// TIA Portal project "practica3_1_3" (V14)

(* hardware
DEVICE "S71500/ET200MP station_1"  S7-1500 station
   slot 0: "Perfil soporte_0"  Rack  6ES7 590-1***0-0AA0
   slot 1: "PLC_1"  CPU 1512C-1 PN  6ES7 512-1CK00-0AB0  V2.1
      slot 3: "Display de la CPU_1"  6ES7591-1AA00-0AA0
DEVICE "PC-System_1"  SIMATIC PC station
   slot 0: "Estación PC SIMATIC"  Rail  SIMATIC PC-Station  V1.0
      slot 125: "Stationmanager"  Station_Manager  V6.0.4
   slot 1: "HMI_RT_1"  WinCC RT Advanced  6AV2 104-0xxxx-xxxx  14.0.0.0
      slot 33792: "Interfaz host"  Host interface
   slot 2: "IE general_1"  IE General  IE_CP  V8.2.0
*)

// ===== PLC "PLC_1"  CPU 1512C-1 PN =====

VAR_GLOBAL   // PLC tag table "Tabla de variables estándar"
   "Tag_1" AT %IW64 : Int;
   "Tag_2" AT %MD100 : Real;
   "PT100" AT %MD102 : Real;
   "setopoint" AT %MW56 : Int;
   "Tag_5" AT %Q4.0 : Bool;
   "Start" AT %M0.0 : Bool;
   "Stop" AT %M0.1 : Bool;
   "activarpid1" AT %M0.2 : Bool;
   "activarpid2" AT %M0.3 : Bool;
   "activarpid3" AT %M0.4 : Bool;
   "activarpid4" AT %M0.5 : Bool;
   "activacion1" AT %M0.6 : Bool;
   "activacion2" AT %M0.7 : Bool;
   "activacion3" AT %M1.0 : Bool;
   "actvacion4" AT %M1.1 : Bool;
   "temp1" AT %MD2 : DInt;
   "rangomaxT1" AT %MD6 : DInt;
   "rangominT1" AT %MD10 : DInt;
   "PT100Dint" AT %MD14 : DInt;
   "temp2" AT %MD18 : DInt;
   "rangomaxT2" AT %MD22 : DInt;
   "rangominT2" AT %MD26 : DInt;
   "temp3" AT %MD30 : DInt;
   "rangomaxT3" AT %MD34 : DInt;
   "rangominT3" AT %MD38 : DInt;
   "temp4" AT %MD42 : DInt;
   "rangomaxT4" AT %MD46 : DInt;
   "rangominT4" AT %MD50 : DInt;
   "auxsecuencia1" AT %MW54 : Int;
   "auxsecuencia2" AT %MW58 : Int;
   "Tag_3" AT %IW6 : Int;
   "Tag_4" AT %IW126 : Int;
   "Tag_6" AT %IW132 : Int;
   "Tag_7" AT %IW134 : Int;
   "Tag_8" AT %MW200 : Int;
END_VAR

DATA_BLOCK "Variables de tiempo"   // DB2
{ S7_Optimized_Access := 'TRUE' }
VERSION : 0.1
   VAR RETAIN
      TiempoP1 : DInt := 1000;
      TiempoP2 : DInt := 1000;
      TiempoP3 : DInt := 1000;
      TiempoP4 : DInt := 1000;
      Tempe_etapa1 : DInt := 20;
      Tempe_etapa2 : DInt := 20;
      Tempe_etapa3 : DInt := 20;
      Tempe_etapa4 : DInt := 20;
   END_VAR
   VAR
      Nombre : String := 'Seleccione la receta';
   END_VAR
BEGIN
END_DATA_BLOCK

DATA_BLOCK "secuencia_DB"   // DB3
{ S7_Optimized_Access := 'TRUE' }
VERSION : 0.1
// stored: InstanceOfName secuencia
"secuencia"
BEGIN
END_DATA_BLOCK

DATA_BLOCK "Reloj"   // DB4
{ S7_Optimized_Access := 'TRUE' }
VERSION : 0.1
   VAR
      Hora_actual : DTL;
   END_VAR
   VAR RETAIN
      Ajustar_hora : DTL;
   END_VAR
   VAR
      Estado_lectura : Word;
      Escribir_hora : Bool;
      Estado_escritura : Word;
   END_VAR
   VAR RETAIN
      Gain_1 : Real;
      Ti : Real;
      Td : Real;
      TdFiltRatio : Real;
      PWeighting : Real;
      DWeighting : Real;
      Cycle : Real;
   END_VAR
BEGIN
END_DATA_BLOCK

FUNCTION_BLOCK "secuencia"   // FB1, GRAPH_PLUS
{ S7_Optimized_Access := 'TRUE' }
VERSION : 0.1
   VAR_INPUT
      OFF_SQ : Bool := false;   // Desactivar cadena
      INIT_SQ : Bool := false;   // Poner cadena en estado inicial
      ACK_EF : Bool := false;   // Acusar todos los errores y fallos
      S_PREV : Bool := false;   // Mostrar la etapa anterior en el parámetro S_NO
      S_NEXT : Bool := false;   // Mostrar la etapa siguiente en el parámetro S_NO
      SW_AUTO : Bool := false;   // Modo automático
      SW_TAP : Bool := false;   // Semiautomático/continuar con transición
      SW_TOP : Bool := false;   // Semiautomático/transición ignorada
      SW_MAN : Bool := false;   // Modo manual
      S_SEL : Int := 0;   // Seleccionar la etapa que debe mostrarse en S_NO
      S_ON : Bool := false;   // Activar la etapa del parámetro S_NO
      S_OFF : Bool := false;   // Desactivar el incremento presente en el parámetro S_NO
      T_PUSH : Bool := false;   // Habilitar conmutación de transición en modo semiautomático
   END_VAR
   VAR_OUTPUT
      S_NO : Int := 0;   // Número de etapa
      S_MORE : Bool := false;   // Existen más etapas que pueden mostrarse en S_NO.
      S_ACTIVE : Bool := false;   // El incremento presente en el parámetro S_NO está activo
      ERR_FLT : Bool := false;   // Error de grupo interlock o supervisión
      AUTO_ON : Bool := false;   // Modo automático activado
      TAP_ON : Bool := false;   // Modo semiautomático/etapa con transición activada
      TOP_ON : Bool := false;   // Modo semiautomático/Ignorar transición activado
      MAN_ON : Bool := false;   // Modo manual activado
   END_VAR
   VAR
      HMI_INFO : Array[0..8] of UInt;
      IF_PAR : G7_IfParPlus_V4;
      RT_DATA : G7_RTDataPlus_V4;   // Área de datos interna
      Trans2 : G7_TransitionPlus_V4;   // Estructura de la transición
      Trans3 : G7_TransitionPlus_V4;   // Estructura de la transición
      Trans4 : G7_TransitionPlus_V4;   // Estructura de la transición
      Trans5 : G7_TransitionPlus_V4;   // Estructura de la transición
      Trans11 : G7_TransitionPlus_V4;   // Estructura de la transición
      Trans12 : G7_TransitionPlus_V4;   // Estructura de la transición
      Trans13 : G7_TransitionPlus_V4;   // Estructura de la transición
      Trans14 : G7_TransitionPlus_V4;   // Estructura de la transición
      Trans15 : G7_TransitionPlus_V4;   // Estructura de la transición
      reposo : G7_StepPlus_V4;   // Estructura de la etapa
      "Etapa 1" : G7_StepPlus_V4;   // Estructura de la etapa
      "Etapa 2" : G7_StepPlus_V4;   // Estructura de la etapa
      "Etapa 3" : G7_StepPlus_V4;   // Estructura de la etapa
      "paso 4" : G7_StepPlus_V4;   // Estructura de la etapa
      "Verificación Sp" : G7_StepPlus_V4;   // Estructura de la etapa
      Verificación_Et2 : G7_StepPlus_V4;   // Estructura de la etapa
      Verificación_Et3 : G7_StepPlus_V4;   // Estructura de la etapa
      "Verificación Et_4" : G7_StepPlus_V4;   // Estructura de la etapa
      SINI : Array[0..1] of USInt;
      LSTT : Array[0..8] of USInt;
      ATAJ : Array[0..8] of USInt;
      ATAB : Array[0..8] of USInt;
      PSTT : Array[0..8] of USInt;
      NSTT : Array[0..8] of USInt;
      ASSJ : Array[0..8] of USInt;
      ASSB : Array[0..8] of USInt;
      PTTS : Array[0..8] of USInt;
      NTTS : Array[0..8] of USInt;
      SW_SQTS : Array[0..8] of USInt;
      SWITCH : Array[0..0] of USInt;
      TVX : Array[0..1] of USInt;
      TTX : Array[0..1] of USInt;
      TSX : Array[0..1] of USInt;
      S00X : Array[0..1] of USInt;
      SOFFX : Array[0..1] of USInt;
      SONX : Array[0..1] of USInt;
      SAX : Array[0..1] of USInt;
      SERRX : Array[0..9] of USInt;
      SMX : Array[0..9] of USInt;
      S0X : Array[0..9] of USInt;
      S1X : Array[0..9] of USInt;
      IL_ALARM_INST : Diag_Alarm;
      SUP_ALARM_INST : Diag_Alarm;
      STEP_TIME_ALARM_INST : Diag_Alarm;
      IEC_TIMER_INST : IEC_TIMER;
   END_VAR
   // SINI[0] := 2;
   // LSTT[0] := 255;
   // LSTT[1] := 255;
   // LSTT[2] := 255;
   // LSTT[8] := 255;
   // ATAJ[1] := 1;
   // ATAJ[2] := 2;
   // ATAJ[3] := 3;
   // ATAJ[4] := 4;
   // ATAJ[5] := 5;
   // ATAJ[6] := 6;
   // ATAJ[7] := 7;
   // ATAJ[8] := 8;
   // ATAB[1] := 1;
   // ATAB[2] := 2;
   // ATAB[3] := 3;
   // NSTT[6] := 2;
   // ATAB[5] := 5;
   // ATAB[6] := 6;
   // ATAB[7] := 7;
   // ATAB[8] := 8;
   // PSTT[1] := 2;
   // PSTT[2] := 3;
   // PSTT[3] := 4;
   // PSTT[8] := 8;
   // PSTT[5] := 5;
   // PSTT[6] := 6;
   // PSTT[7] := 7;
   // NSTT[5] := 1;
   // NSTT[0] := 6;
   // NSTT[1] := 7;
   // NSTT[2] := 8;
   // NSTT[8] := 4;
   // ASSJ[1] := 1;
   // ASSJ[2] := 2;
   // ASSJ[3] := 3;
   // ASSJ[4] := 4;
   // ASSB[1] := 1;
   // ASSB[2] := 2;
   // ASSB[3] := 3;
   // ASSB[4] := 4;
   // PTTS[0] := 255;
   // PTTS[5] := 4;
   // PTTS[3] := 7;
   // PTTS[4] := 8;
   // NTTS[5] := 5;
   // NTTS[2] := 1;
   // NTTS[3] := 2;
   // NTTS[4] := 3;
   // TVX[0] := 16#1;
   // TTX[0] := 16#1;
   // TSX[0] := 16#1;
   // S00X[0] := 16#1;
   // SOFFX[0] := 16#1;
   // SONX[0] := 16#1;
   // SAX[0] := 16#1;
   // SERRX[0] := 16#1;
   // SMX[0] := 16#1;
   // S0X[0] := 16#1;
   // S1X[0] := 16#1;
   // LSTT[4] := 255;
   // NSTT[7] := 3;
   // ATAB[4] := 4;
   // PSTT[0] := 1;
   // NSTT[4] := 5;
   // ASSJ[5] := 5;
   // ASSB[5] := 5;
   // PTTS[1] := 5;
   // NTTS[0] := 4;
   // LSTT[5] := 255;
   // LSTT[6] := 255;
   // LSTT[7] := 255;
   // ASSJ[6] := 6;
   // ASSJ[7] := 7;
   // ASSJ[8] := 8;
   // ASSB[6] := 6;
   // ASSB[7] := 7;
   // ASSB[8] := 8;
   // PTTS[2] := 6;
   // PTTS[7] := 1;
   // PTTS[8] := 2;
   // NTTS[6] := 6;
   // NTTS[7] := 7;
   // NTTS[8] := 8;
BEGIN
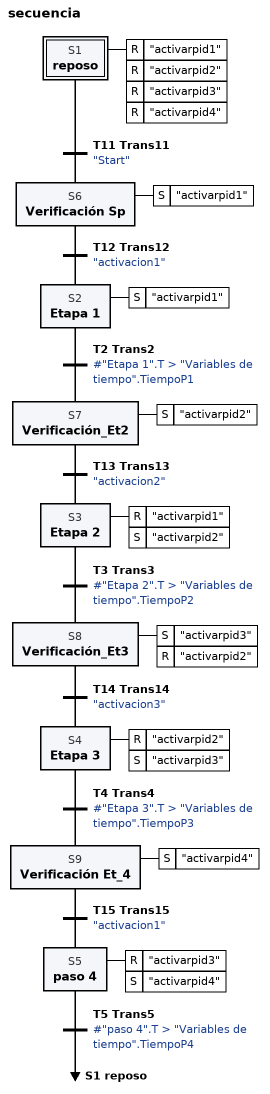
   // sequencer 1
   INITIAL_STEP reposo:   // S1, max time T#10S, warning time T#7S
              R    "activarpid1"
              R    "activarpid2"
              R    "activarpid3"
              R    "activarpid4"
   END_STEP
   TRANSITION Trans11 FROM reposo TO "Verificación Sp"   // T11
      := "Start";
   END_TRANSITION
   STEP "Etapa 1":   // S2, max time T#10S, warning time T#7S
              S    "activarpid1"
   END_STEP
   TRANSITION Trans2 FROM "Etapa 1" TO Verificación_Et2   // T2
      := #"Etapa 1".T > "Variables de tiempo".TiempoP1;
   END_TRANSITION
   STEP "Etapa 2":   // S3, max time T#10S, warning time T#7S
              R    "activarpid1"
              S    "activarpid2"
   END_STEP
   TRANSITION Trans3 FROM "Etapa 2" TO Verificación_Et3   // T3
      := #"Etapa 2".T > "Variables de tiempo".TiempoP2;
   END_TRANSITION
   STEP "Etapa 3":   // S4, max time T#10S, warning time T#7S
              R    "activarpid2"
              S    "activarpid3"
   END_STEP
   TRANSITION Trans4 FROM "Etapa 3" TO "Verificación Et_4"   // T4
      := #"Etapa 3".T > "Variables de tiempo".TiempoP3;
   END_TRANSITION
   STEP "paso 4":   // S5, max time T#10S, warning time T#7S
              R    "activarpid3"
              S    "activarpid4"
   END_STEP
   TRANSITION Trans5 FROM "paso 4" TO reposo   // T5, jump
      := #"paso 4".T > "Variables de tiempo".TiempoP4;
   END_TRANSITION
   STEP "Verificación Sp":   // S6, max time T#10S, warning time T#7S
              S    "activarpid1"
   END_STEP
   TRANSITION Trans12 FROM "Verificación Sp" TO "Etapa 1"   // T12
      := "activacion1";
   END_TRANSITION
   STEP Verificación_Et2:   // S7, max time T#10S, warning time T#7S
              S    "activarpid2"
   END_STEP
   TRANSITION Trans13 FROM Verificación_Et2 TO "Etapa 2"   // T13
      := "activacion2";
   END_TRANSITION
   STEP Verificación_Et3:   // S8, max time T#10S, warning time T#7S
              S    "activarpid3"
              R    "activarpid2"
   END_STEP
   TRANSITION Trans14 FROM Verificación_Et3 TO "Etapa 3"   // T14
      := "activacion3";
   END_TRANSITION
   STEP "Verificación Et_4":   // S9, max time T#10S, warning time T#7S
              S    "activarpid4"
   END_STEP
   TRANSITION Trans15 FROM "Verificación Et_4" TO "paso 4"   // T15
      := "activacion1";
   END_TRANSITION
END_FUNCTION_BLOCK

FUNCTION "normalizar_temp" : Void   // FC1, LAD
{ S7_Optimized_Access := 'TRUE' }
VERSION : 0.1
BEGIN

REGION Network 1: Ajuste de los datos de entrada
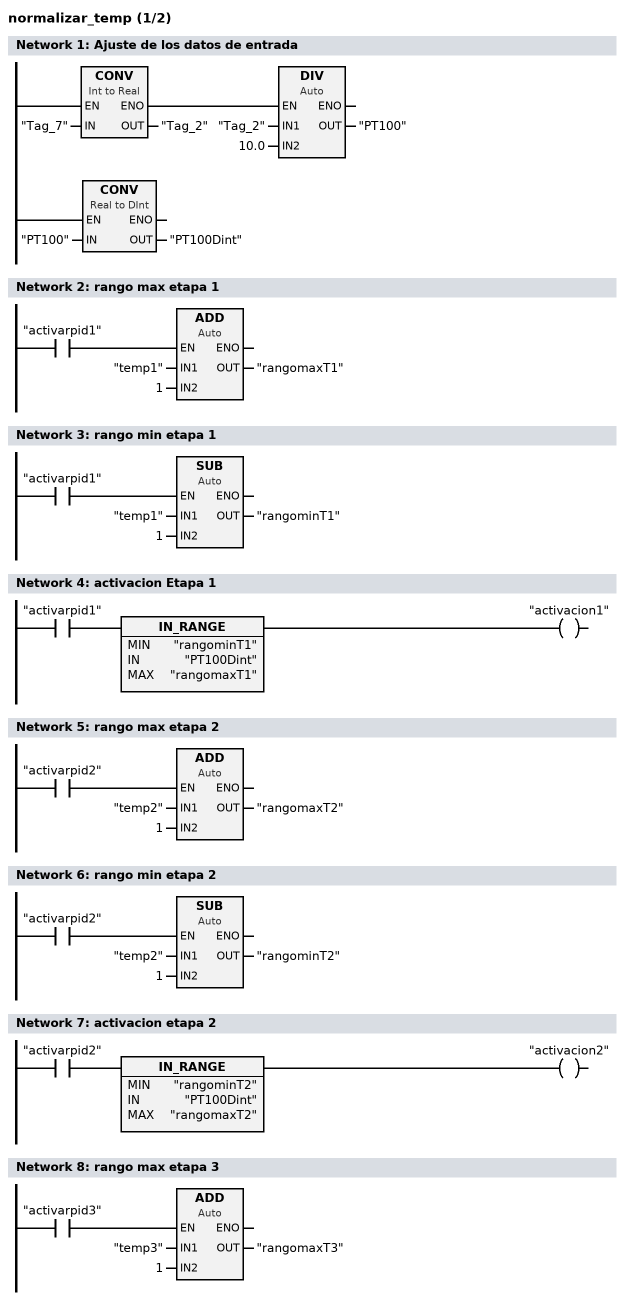
   RUNG wire#powerrail
      { S7_Templates := "[SrcType := Int, DestType := Real]" } Convert(in := "Tag_7", out => "Tag_2")
      Div(in1 := "Tag_2", in2 := 10.0, out => "PT100")
   END_RUNG
   RUNG wire#powerrail
      { S7_Templates := "[SrcType := Real, DestType := DInt]" } Convert(in := "PT100", out => "PT100Dint")
   END_RUNG
   // the same network as SCL:
   "Tag_2" := INT_TO_REAL("Tag_7");
   "PT100" := "Tag_2" / 10.0;
   "PT100Dint" := REAL_TO_DINT("PT100");
END_REGION

REGION Network 2: rango max etapa 1
   RUNG wire#powerrail
      Contact( "activarpid1" )
      Add(in1 := "temp1", in2 := 1, out => "rangomaxT1")
   END_RUNG
   // the same network as SCL:
   IF "activarpid1" THEN "rangomaxT1" := "temp1" + 1; END_IF;
END_REGION

REGION Network 3: rango min etapa 1
   RUNG wire#powerrail
      Contact( "activarpid1" )
      Sub(in1 := "temp1", in2 := 1, out => "rangominT1")
   END_RUNG
   // the same network as SCL:
   IF "activarpid1" THEN "rangominT1" := "temp1" - 1; END_IF;
END_REGION

REGION Network 4: activacion Etapa 1
   RUNG wire#powerrail
      Contact( "activarpid1" )
      { S7_Templates := "SrcType := DInt" } InRange(min := "rangominT1", in := "PT100Dint", max := "rangomaxT1")
      Coil( "activacion1" )
   END_RUNG
   // the same network as SCL:
   "activacion1" := "activarpid1" AND ("rangominT1" <= "PT100Dint") AND ("PT100Dint" <= "rangomaxT1");
END_REGION

REGION Network 5: rango max etapa 2
   RUNG wire#powerrail
      Contact( "activarpid2" )
      Add(in1 := "temp2", in2 := 1, out => "rangomaxT2")
   END_RUNG
   // the same network as SCL:
   IF "activarpid2" THEN "rangomaxT2" := "temp2" + 1; END_IF;
END_REGION

REGION Network 6: rango min etapa 2
   RUNG wire#powerrail
      Contact( "activarpid2" )
      Sub(in1 := "temp2", in2 := 1, out => "rangominT2")
   END_RUNG
   // the same network as SCL:
   IF "activarpid2" THEN "rangominT2" := "temp2" - 1; END_IF;
END_REGION

REGION Network 7: activacion etapa 2
   RUNG wire#powerrail
      Contact( "activarpid2" )
      { S7_Templates := "SrcType := DInt" } InRange(min := "rangominT2", in := "PT100Dint", max := "rangomaxT2")
      Coil( "activacion2" )
   END_RUNG
   // the same network as SCL:
   "activacion2" := "activarpid2" AND ("rangominT2" <= "PT100Dint") AND ("PT100Dint" <= "rangomaxT2");
END_REGION

REGION Network 8: rango max etapa 3
   RUNG wire#powerrail
      Contact( "activarpid3" )
      Add(in1 := "temp3", in2 := 1, out => "rangomaxT3")
   END_RUNG
   // the same network as SCL:
   IF "activarpid3" THEN "rangomaxT3" := "temp3" + 1; END_IF;
END_REGION

REGION Network 9: rango min paso 3
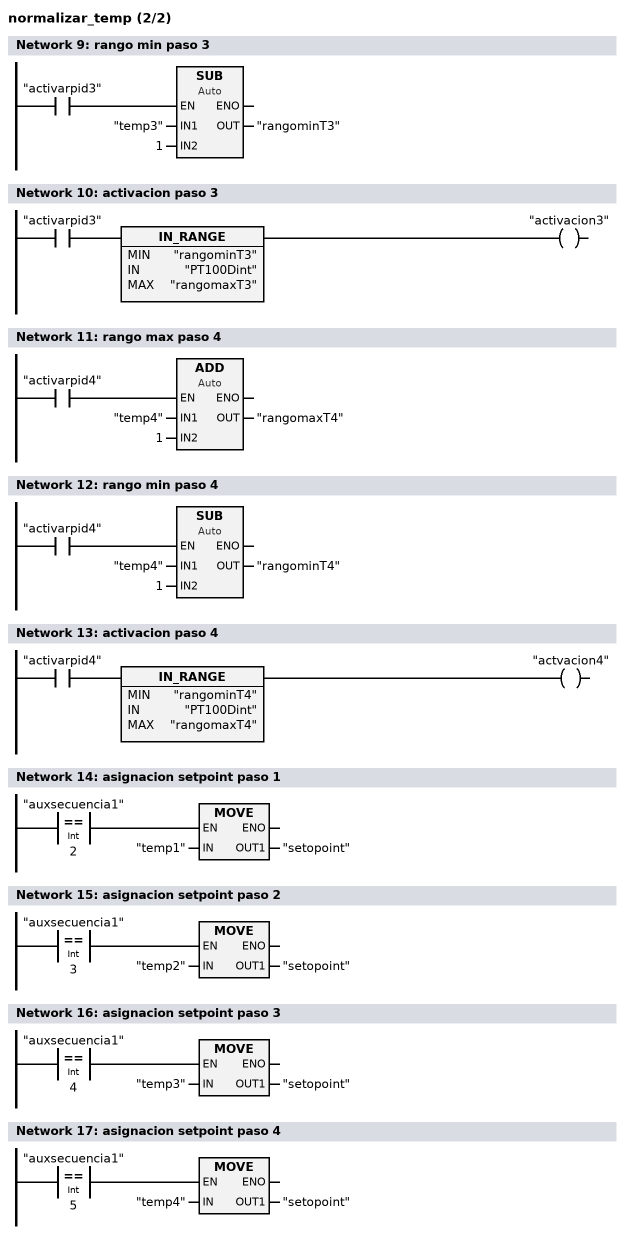
   RUNG wire#powerrail
      Contact( "activarpid3" )
      Sub(in1 := "temp3", in2 := 1, out => "rangominT3")
   END_RUNG
   // the same network as SCL:
   IF "activarpid3" THEN "rangominT3" := "temp3" - 1; END_IF;
END_REGION

REGION Network 10: activacion paso 3
   RUNG wire#powerrail
      Contact( "activarpid3" )
      { S7_Templates := "SrcType := DInt" } InRange(min := "rangominT3", in := "PT100Dint", max := "rangomaxT3")
      Coil( "activacion3" )
   END_RUNG
   // the same network as SCL:
   "activacion3" := "activarpid3" AND ("rangominT3" <= "PT100Dint") AND ("PT100Dint" <= "rangomaxT3");
END_REGION

REGION Network 11: rango max paso 4
   RUNG wire#powerrail
      Contact( "activarpid4" )
      Add(in1 := "temp4", in2 := 1, out => "rangomaxT4")
   END_RUNG
   // the same network as SCL:
   IF "activarpid4" THEN "rangomaxT4" := "temp4" + 1; END_IF;
END_REGION

REGION Network 12: rango min paso 4
   RUNG wire#powerrail
      Contact( "activarpid4" )
      Sub(in1 := "temp4", in2 := 1, out => "rangominT4")
   END_RUNG
   // the same network as SCL:
   IF "activarpid4" THEN "rangominT4" := "temp4" - 1; END_IF;
END_REGION

REGION Network 13: activacion paso 4
   RUNG wire#powerrail
      Contact( "activarpid4" )
      { S7_Templates := "SrcType := DInt" } InRange(min := "rangominT4", in := "PT100Dint", max := "rangomaxT4")
      Coil( "actvacion4" )
   END_RUNG
   // the same network as SCL:
   "actvacion4" := "activarpid4" AND ("rangominT4" <= "PT100Dint") AND ("PT100Dint" <= "rangomaxT4");
END_REGION

REGION Network 14: asignacion setpoint paso 1
   RUNG wire#powerrail
      { S7_Templates := "SrcType := Int" } EQ_Contact(in1 := "auxsecuencia1", in2 := 2)
      Move(in := "temp1", out1 => "setopoint")
   END_RUNG
   // the same network as SCL:
   IF "auxsecuencia1" = 2 THEN "setopoint" := "temp1"; END_IF;
END_REGION

REGION Network 15: asignacion setpoint paso 2
   RUNG wire#powerrail
      { S7_Templates := "SrcType := Int" } EQ_Contact(in1 := "auxsecuencia1", in2 := 3)
      Move(in := "temp2", out1 => "setopoint")
   END_RUNG
   // the same network as SCL:
   IF "auxsecuencia1" = 3 THEN "setopoint" := "temp2"; END_IF;
END_REGION

REGION Network 16: asignacion setpoint paso 3
   RUNG wire#powerrail
      { S7_Templates := "SrcType := Int" } EQ_Contact(in1 := "auxsecuencia1", in2 := 4)
      Move(in := "temp3", out1 => "setopoint")
   END_RUNG
   // the same network as SCL:
   IF "auxsecuencia1" = 4 THEN "setopoint" := "temp3"; END_IF;
END_REGION

REGION Network 17: asignacion setpoint paso 4
   RUNG wire#powerrail
      { S7_Templates := "SrcType := Int" } EQ_Contact(in1 := "auxsecuencia1", in2 := 5)
      Move(in := "temp4", out1 => "setopoint")
   END_RUNG
   // the same network as SCL:
   IF "auxsecuencia1" = 5 THEN "setopoint" := "temp4"; END_IF;
END_REGION
END_FUNCTION

FUNCTION "Lectura hora" : Void   // FC2, LAD
{ S7_Optimized_Access := 'TRUE' }
VERSION : 0.1
BEGIN

REGION Network 1: leer hora
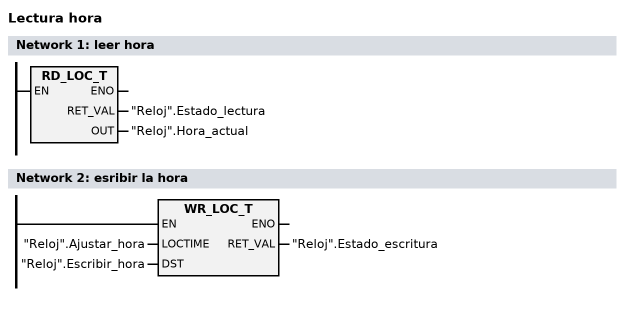
   "Reloj".Estado_lectura := RD_LOC_T(OUT => "Reloj".Hora_actual);
END_REGION

REGION Network 2: esribir la hora
   "Reloj".Estado_escritura := WR_LOC_T(LOCTIME := "Reloj".Ajustar_hora, DST := "Reloj".Escribir_hora);
END_REGION
END_FUNCTION

ORGANIZATION_BLOCK "Main"   // OB1, LAD, ProgramCycle
TITLE = "Main Program Sweep (Cycle)"
{ S7_Optimized_Access := 'TRUE' }
VERSION : 0.1
   VAR_INPUT
      Initial_Call : Bool;   // Initial call of this OB
      Remanence : Bool;   // =True, if remanent data are available
   END_VAR
BEGIN

REGION Network 1
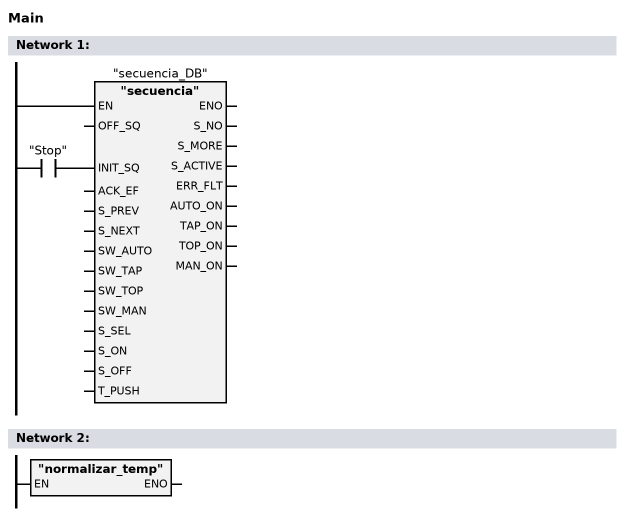
   RUNG wire#powerrail
      "secuencia_DB"(INIT_SQ := wire#w1, OFF_SQ :=, ACK_EF :=, S_PREV :=, S_NEXT :=, SW_AUTO :=, SW_TAP :=, SW_TOP :=, SW_MAN :=, S_SEL :=, S_ON :=, S_OFF :=, T_PUSH :=, S_NO =>, S_MORE =>, S_ACTIVE =>, ERR_FLT =>, AUTO_ON =>, TAP_ON =>, TOP_ON =>, MAN_ON =>)
   END_RUNG
   RUNG wire#powerrail
      Contact( "Stop" )
   END_RUNG wire#w1
   // the same network as SCL:
   "secuencia_DB"(INIT_SQ := "Stop");   // "secuencia"
END_REGION

REGION Network 2
   RUNG wire#powerrail
      "normalizar_temp"()
   END_RUNG
   // the same network as SCL:
   "normalizar_temp"();
END_REGION
END_ORGANIZATION_BLOCK

ORGANIZATION_BLOCK "Cyclic interrupt"   // OB30, LAD, CyclicInterrupt
{ S7_Optimized_Access := 'TRUE' }
VERSION : 0.1
   VAR_INPUT
      Initial_Call : Bool;   // Initial call of this OB
      Event_Count : Int;   // Events discarded
   END_VAR
BEGIN

REGION Network 1
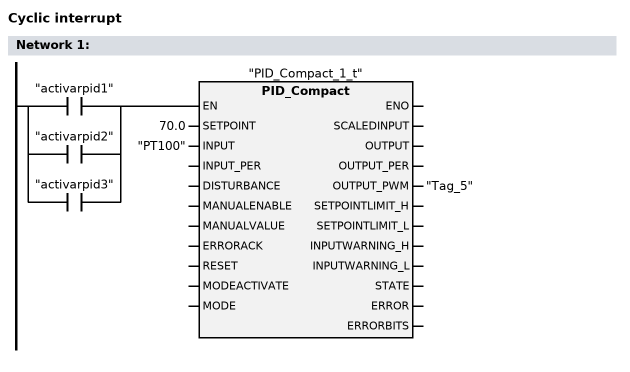
   IF "activarpid1" OR "activarpid2" OR "activarpid3" THEN
       "PID_Compact_1_t"(Setpoint := 70.0, Input := "PT100", Output_PWM => "Tag_5");   // PID_Compact
   END_IF;
END_REGION
END_ORGANIZATION_BLOCK

(* ===== HMI "HMI_RT_1" =====
system functions are stored by id; their names below are inferred from use
connection "HMI_Conexión_1": ETHERNET, S7_1500_OMS
connection "HMI_Conexión_2": ETHERNET, S7_1500_OMS

HMI tags "Tabla de variables estándar"
   "Start" : Bool = PLC Start AT %M0.0, 1 s
   "temp1" : DInt = PLC temp1 AT %MD2, 1 s
   "temp2" : DInt = PLC temp2 AT %MD18, 1 s
   "temp3" : DInt = PLC temp3 AT %MD30, 1 s
   "temp4" : DInt = PLC temp4 AT %MD42, 1 s
   "Variables de tiempo_TiempoP1" : DInt = PLC "Variables de tiempo".TiempoP1, 1 s
   "Variables de tiempo_TiempoP2" : DInt = PLC "Variables de tiempo".TiempoP2, 1 s
   "Variables de tiempo_TiempoP3" : DInt = PLC "Variables de tiempo".TiempoP3, 1 s
   "Variables de tiempo_TiempoP4" : DInt = PLC "Variables de tiempo".TiempoP4, 1 s
   "Stop" : Bool = PLC Stop AT %M0.1, 1 s
   "Reloj_Hora_actual" : DTL = PLC Reloj.Hora_actual, 1 s
   "Reloj_Ajustar_hora" : DTL = PLC Reloj.Ajustar_hora, 1 s
   "Variables de tiempo_Nombre" : String[254] = PLC "Variables de tiempo".Nombre, 1 s
   "Variables de tiempo_Tempe_etapa1" : DInt = PLC "Variables de tiempo".Tempe_etapa1, 1 s
   "Variables de tiempo_Tempe_etapa2" : DInt = PLC "Variables de tiempo".Tempe_etapa2, 1 s
   "Variables de tiempo_Tempe_etapa3" : DInt = PLC "Variables de tiempo".Tempe_etapa3, 1 s
   "Variables de tiempo_Tempe_etapa4" : DInt = PLC "Variables de tiempo".Tempe_etapa4, 1 s

recipe "Pandebono": Nombre <- "Variables de tiempo_Nombre", Tiempo etapa1(miliseg) <- "Variables de tiempo_TiempoP1", Temperatura_et1(°C) <- "Variables de tiempo_Tempe_etapa1", Tiempo etapa2(miliseg) <- "Variables de tiempo_TiempoP2", Temperatura_et2(°C) <- "Variables de tiempo_Tempe_etapa2", Tiempo etapa3(miliseg) <- "Variables de tiempo_TiempoP3", Temperatura_et3(°C) <- "Variables de tiempo_Tempe_etapa3", Tiempo etapa4(miliseg) <- "Variables de tiempo_TiempoP4", Temperatura_et4(°C) <- "Variables de tiempo_Tempe_etapa4"

screen "Imagen_1" 1440x900
   Button "Botón_1" at 284,97 size 131x45; TextOff 'start'
      on Press: SetBit("Start")
      on Release: ResetBit("Start")
   IOField "Campo ES_1" at 457,97 size 96x32; FormatPattern 99; Unit °C
      ProcessValue <- "temp1"
   IOField "Campo ES_2" at 457,143 size 96x32; FormatPattern 99; Unit °C
      ProcessValue <- "temp2"
   IOField "Campo ES_3" at 457,189 size 96x32; FormatPattern 99; Unit °C
      ProcessValue <- "temp3"
   IOField "Campo ES_4" at 457,235 size 96x32; FormatPattern 99; Unit °C
      ProcessValue <- "temp4"
   IOField "Campo ES_5" at 654,96 size 96x32; FormatPattern 99; Unit s
      ProcessValue <- "Variables de tiempo_TiempoP1"
   IOField "Campo ES_6" at 654,142 size 96x32; FormatPattern 99; Unit s
      ProcessValue <- "Variables de tiempo_TiempoP2"
   IOField "Campo ES_7" at 655,189 size 96x32; FormatPattern 99; Unit s
      ProcessValue <- "Variables de tiempo_TiempoP3"
   IOField "Campo ES_8" at 655,235 size 96x32; FormatPattern 99; Unit s
      ProcessValue <- "Variables de tiempo_TiempoP4"
   TextField "Campo de texto_1" at 553,106 size 65x22; Text 'Temp_1'
   TextField "Campo de texto_2" at 554,153 size 65x22; Text 'Temp_2'
   TextField "Campo de texto_3" at 555,200 size 65x22; Text 'Temp_3'
   TextField "Campo de texto_4" at 556,247 size 65x22; Text 'Temp_4'
   TextField "Campo de texto_5" at 753,105 size 79x22; Text 'Tiempo_1'
   TextField "Campo de texto_6" at 753,153 size 79x22; Text 'Tiempo_2'
   TextField "Campo de texto_7" at 753,201 size 79x22; Text 'Tiempo_3'
   TextField "Campo de texto_8" at 753,249 size 79x22; Text 'Tiempo_4'
   Button "Botón_2" at 284,170 size 131x45; TextOff 'Stop'
      on Release: ResetBit("Stop")
      on Press: SetBit("Stop")
   Button "Botón_3" at 450,361 size 326x32; TextOff 'Cambiar'; Authorization "Cambiar_hora"
   TextField "Campo de texto_9" at 449,308 size 104x40; Text 'Hora_actual Hora_ajustar'
   IOField "Campo ES_9" at 579,295 size 194x32; FormatPattern 9999999999999999999999999999999999999999
      ProcessValue <- "Reloj_Hora_actual"
   IOField "Campo ES_10" at 581,323 size 192x32; FormatPattern 9999999999999999999999999999999999999999
      ProcessValue <- "Reloj_Ajustar_hora"
   RecipeView "Visor de recetas_1" at 0,129 size 400x350
*)